{attribute addProperty BoxType "ER3184-0002-0021"}
{attribute addProperty Id "AI_Standard_ChannelAT %I*ARRAY[0..3] OF AI_Standard_Channel_087F71C7128160WcStateAT %I*WcState_F855686C1620InfoDataAT %I*InfoData_BC63D37F80100"}
{attribute addProperty CRC "3082647473"}
{attribute addProperty SizeInBites "224"}
{attribute addProperty SizeInBytes "28"}
TYPE ER3184_83515A0D :
STRUCT
	{attribute addProperty Name "AI_Standard_Channel"}
	AI_Standard_Channel : ARRAY[0..3] OF AI_Standard_Channel_087F71C7;
	{attribute addProperty Name "WcState"}
	WcState : WcState_F855686C;
	{attribute addProperty Name "InfoData"}
	InfoData : InfoData_BC63D37F;
END_STRUCT
END_TYPE

(* stored: Version 1.2.0.0, ProductVersion 3.1.4024.9
   DUT ER3184_83515A0D: Id {9bc1b9fc-80b3-4d0d-9c51-61187bc5aed1} *)
